// TIA Portal project "SWL SEMAFORO 2" (V11)

(* hardware
DEVICE "S7300/ET200 station_1"  SIMATIC 300-Station
   slot 0: "Perfil soporte_0"  Rail  6ES7 390-1***0-0AA0
   slot 2: "PLC_1"  CPU 313C-2 DP  6ES7 313-6CF03-0AB0  V2.6
      slot 0: "Interfaz MPI_1"  MPI
      slot 1: "Interfaz DP_1"  DP
      slot 2: "DI16/DO16_1"  DI16/DO16
      slot 4: "Contaje_1"  Counter
*)

// ===== PLC "PLC_1"  CPU 313C-2 DP =====

VAR_GLOBAL   // PLC tag table "Tabla de variables estándar"
   "PULSADOR" AT %E0.0 : Bool;
   "VERDE COCHES" AT %A0.0 : Bool;
   "AMBAR COCHES" AT %A0.1 : Bool;
   "ROJO COCHES" AT %A0.2 : Bool;
   "ROJO PEATONES" AT %A0.3 : Bool;
   "VERDE PEATONES" AT %A0.4 : Bool;
   "MARCA CICLO" AT %M100.5 : Bool;
   "Tag_3" AT %M10.0 : Bool;
   "Tag_11" AT %M11.0 : Bool;
   "Tag_12" AT %M11.1 : Bool;
   "Tag_13" AT %M10.1 : Bool;
   "CONTADOR" AT %MW20 : Int;
   "CONTROL" AT %MB0 : Byte;
   "Tag_16" AT %M0.0 : Bool;
   "Tag_1" AT %M0.1 : Bool;
   "Tag_4" AT %M0.2 : Bool;
   "Tag_5" AT %M0.3 : Bool;
   "Tag_9" AT %M0.4 : Bool;
   "Tag_10" AT %M30.0 : Bool;
   "Tag_17" AT %M10.2 : Bool;
END_VAR

ORGANIZATION_BLOCK "Main"   // OB1, STL
TITLE = "Main Program Sweep (Cycle)"
{ S7_Optimized_Access := 'FALSE' }
VERSION : 0.1
   VAR_TEMP
      OB1_EV_CLASS : Byte;   // Bits 0-3 = 1 (Coming event), Bits 4-7 = 1 (Event class 1)
      OB1_SCAN_1 : Byte;   // 1 (Cold restart scan 1 of OB 1), 3 (Scan 2-n of OB 1)
      OB1_PRIORITY : Byte;   // Priority of OB Execution
      OB1_OB_NUMBR : Byte;   // 1 (Organization block 1, OB1)
      OB1_RESERVED_1 : Byte;   // Reserved for system
      OB1_RESERVED_2 : Byte;   // Reserved for system
      OB1_PREV_CYCLE : Int;   // Cycle time of previous OB1 scan (milliseconds)
      OB1_MIN_CYCLE : Int;   // Minimum cycle time of OB1 (milliseconds)
      OB1_MAX_CYCLE : Int;   // Maximum cycle time of OB1 (milliseconds)
      OB1_DATE_TIME : Date_And_Time;   // Date and time OB1 started
   END_VAR
BEGIN
END_ORGANIZATION_BLOCK